TYPE Vec4b : ARRAY[1..4] OF BOOL; END_TYPE

(* stored: Version 1.1.0.1, ProductVersion 3.1.4024.12
   DUT Vec4b: Id {f34f7bf4-b6d4-4400-8ccf-14ccf46b1d9e} *)
